Universal Robots PolyScope program: ATI_example_Sanding.urp

Program ATI_example_Sanding (installation=default directory=/programs/usbdisk/20220721 createdIn=3.1.18024.0 lastSavedIn=3.15.6.106324 robotSerialNumber=2016353406)
Calibrated DH parameters: a=[0.000241, -0.156882, -0.391168, -0.000034, 0.000033, 0]; d=[0.08909, 1210.353649, -1202.089359, -8.154207, 0.094912, 0.082482]; alpha=[1.570962, 0.000326, -0.003342, 1.570446, -1.570439, 0]; deltaTheta=[0.000082, 1.192638, -1.263181, 0.0705, 0.00007, 0.000052]
BeforeStart
  Folder Move to Initial start position
    'Set Actual Robot Payload (enter your TCP payload)'
    Script: set_payload(1)
    'Move to a Start Position (reteach this point to a safe home location!)'
    MoveJ speed 60 deg/s, acceleration 80 deg/s^2 (useActiveTCP=false)
      Waypoint Start: 
    Wait Sleep waitTime=0.01
    URCap F/T Sensor Command (ATI Axia Force/Torque Sensor, ATI Industrial Automation) dataModel(WEIGHT=0.025, running=Enable)
    'Use Options to adjust Filter for your sander vibrations'
    URCap F/T Sensor Options (ATI Axia Force/Torque Sensor, ATI Industrial Automation) dataModel(STATUS=80000008, LOGGING_LEVEL=0, FILTER=4)
    'Adjust sensitivity of UR Force mode'
    Script: force_mode_set_damping(1)
    Script: force_mode_set_gain_scaling(.5)
Robot Program (runOnlyOnce=false)
  Folder Bias the sensor
    Wait Sleep waitTime=1
    URCap F/T Sensor Command (ATI Axia Force/Torque Sensor, ATI Industrial Automation) dataModel(running=Bias)
  Folder Move down until the tool touches a surface
    MoveJ speed 60 deg/s, acceleration 80 deg/s^2 (useActiveTCP=true)
      'Move to hover above surface (reteach to a point ~5cm above surface)'
      Waypoint AboveTable: 
    If ATI_ZForce>-2 (checkContinuously=true)
      'Relative motion in Z'
      Script: movel(pose_trans(get_actual_tcp_pose(),p[0,0,.2,0,0,0]),a=0.05,v=.04,t=0,r=0)
  Folder Move across the surface while applying 2N of force
    Force Simple feature=Joint_6_name; selection=[0, 0, 1, 0, 0, 0]; wrench=[0, 0, 2, 0, 0, 0]; limitsForce=[0.15, 0.15, 0.15, 1.047198, 1.047198, 1.047198]; limitsMotion=[0.1, 0.1, 0.1, 0.349066, 0.349066, 0.349066]
      Folder If the tool encounters too much resistance, return to start position
        If xyPlaneForce <20 (checkContinuously=true)
          'Relative motion 0.3m in -Y'
          Script: movel(pose_trans(get_actual_tcp_pose(), p[0,-.3,0,0,0,0]),a=0.04,v=.02,t=0,r=0)
  Folder Reset to a start position
    'Relative motion in Z'
    Script: movel(pose_trans(get_actual_tcp_pose(), p[0,0,-.2,0,0,0]),a=0.04,v=.1,t=0,r=0)
  Folder Move down until the tool touchs a surface
    If ATI_ZForce>-2 (checkContinuously=true)
      'Relative motion in Z'
      Script: movel(pose_trans(get_actual_tcp_pose(),p[0,0,.2,0,0,0]),a=0.05,v=.04,t=0,r=0)
  Folder Move across the surface while applying 2N of force
    Force Simple feature=Joint_6_name; selection=[0, 0, 1, 0, 0, 0]; wrench=[0, 0, 2, 0, 0, 0]; limitsForce=[0.15, 0.15, 0.15, 1.047198, 1.047198, 1.047198]; limitsMotion=[0.1, 0.1, 0.1, 0.349066, 0.349066, 0.349066]
      Folder If the tool encounters too much resistance, return to start position
        If xyPlaneForce <20 (checkContinuously=true)
          'Relative motion 0.3m in +Y'
          Script: movel(pose_trans(get_actual_tcp_pose(), p[0,.3,0,0,0,0]),a=0.04,v=.02,t=0,r=0)
  Folder Reset to a start position
    Script: movel(pose_trans(get_actual_tcp_pose(), p[0,0,-.2,0,0,0]),a=0.04,v=.1,t=0,r=0)
    MoveJ speed 60 deg/s, acceleration 80 deg/s^2 (useActiveTCP=true)
      Waypoint Start: 
Thread Thread_1 (runOnlyOnce=false)
  'UR Command get_tcp_force() is transformed to Base'
  TCPForce := get_tcp_force()
  'ATI reading in the sensor frame'
  ATI_rawFT := ati_ftsensor.get_raw_ft()
  'Adjust the TCP offset parameters for your tool!'
  'ATI reading in the TCP frame: TCP is .5m offset in Z from the sensor measuring face'
  ATI_TCP_FT := ati_ftsensor.get_tcp_ft(0, 0, .5, 0, 0, 0)
  ATI_ZForce := ATI_TCP_FT[2]
  Folder Get magnitude of force in X-Y plane, accounting for friction of tool
    xyPlaneForce := sqrt(pow(TCPForce[0], 2) + pow(TCPForce[1], 2)) - 0.3*ATI_ZForce
  Wait Sleep waitTime=0.01
